Fanuc KAREL source: compact_preamble.KL

PROGRAM NC0002
%NOLOCKGROUP
ROUTINE R
VAR
S1:INTEGER
BEGIN
S1=1
IF (S1=1) THEN
S1=(S1 + 1)
ELSE
S1=(S1 + 2)
ENDIF
END R
BEGIN
R
END NC0002
